// TIA Portal V20 export
FUNCTION_BLOCK "SysSensor"   // FB2040, FBD
TITLE = manage a sensor
{ S7_Optimized_Access := 'TRUE' }
AUTHOR : MiCROTEC
VERSION : 1.5
// -2021.12 : Martin / -2018.12 : Martin
// stored: AutoNumber false, MemoryReserve 100, SetENOAutomatically false
   VAR_INPUT
      errOccIn { ExternalAccessible := 'False'; ExternalVisible := 'False'; ExternalWritable := 'False'} : Bool;   // fault input (sensor signal or a combination of sensors)
      errOccVal { ExternalAccessible := 'False'; ExternalVisible := 'False'; ExternalWritable := 'False'} : Real;   // fault value for fault input
      errFreeIn { ExternalAccessible := 'False'; ExternalVisible := 'False'; ExternalWritable := 'False'} : Bool;   // fault input 2 (sensor signal or a combination of sensors)
      errFreeVal { ExternalAccessible := 'False'; ExternalVisible := 'False'; ExternalWritable := 'False'} : Real;   // fault value for fault input 2
      errCycleIn { ExternalAccessible := 'False'; ExternalVisible := 'False'; ExternalWritable := 'False'} : Bool;   // fault cycle input (this input increment a counter, counter is reset with rise or fallinge edge of sensor )
      errCycleVal { ExternalAccessible := 'False'; ExternalVisible := 'False'; ExternalWritable := 'False'} : Real;   // fault cycle value (if counter exceeds this value then error is set )
      sensor { ExternalAccessible := 'False'; ExternalVisible := 'False'; ExternalWritable := 'False'} : Bool;   // sensor signal
      enable { ExternalAccessible := 'False'; ExternalVisible := 'False'; ExternalWritable := 'False'} : Bool;   // if enable is true than the counter count, ex. run message from conv.
      ack { ExternalAccessible := 'False'; ExternalVisible := 'False'; ExternalWritable := 'False'} : Bool;   // acknowledg faults
      onDelVal { ExternalAccessible := 'False'; ExternalVisible := 'False'; ExternalWritable := 'False'} : Real;   // delayed on value for delayed on
      offDelVal { ExternalAccessible := 'False'; ExternalVisible := 'False'; ExternalWritable := 'False'} : Real;   // delayed off value for delayed off
      occOnVal { ExternalAccessible := 'False'; ExternalVisible := 'False'; ExternalWritable := 'False'} : Real;   // delayed on value for sensor occupied
      occOffVal { ExternalAccessible := 'False'; ExternalVisible := 'False'; ExternalWritable := 'False'} : Real;   // delayed off value for sensor occupied
      cntrVal { ExternalAccessible := 'False'; ExternalVisible := 'False'; ExternalWritable := 'False'} : Real;   // count value per cycle, if absolut encoder than activate "Param.AbsolutEncoder"
      absEnc { ExternalAccessible := 'False'; ExternalVisible := 'False'; ExternalWritable := 'False'} : Bool;   // activate absolut encoder for "countValue"
      reset { ExternalAccessible := 'False'; ExternalVisible := 'False'; ExternalWritable := 'False'} : Bool;   // reset the counter values and also the outputs
   END_VAR
   VAR_OUTPUT
      err { ExternalAccessible := 'False'; ExternalVisible := 'False'; ExternalWritable := 'False'} : Bool;   // Sensor fault , sensor is broken or is dirty
      errOcc { ExternalAccessible := 'False'; ExternalVisible := 'False'; ExternalWritable := 'False'} : Bool;   // Sensor fault , was to long occupied, maybe dirty or misaligned
      errFree { ExternalAccessible := 'False'; ExternalVisible := 'False'; ExternalWritable := 'False'} : Bool;   // Sensor fault , was to long free, maybe dirty or misaligned
      errCycle { ExternalAccessible := 'False'; ExternalVisible := 'False'; ExternalWritable := 'False'} : Bool;   // Sensor fault , plausibility check of cycles, after a certain amount(#errCycleVal) of trigger(#errCycleIn) the sensor had no rising or falling edge
      onDel { ExternalAccessible := 'False'; ExternalVisible := 'False'; ExternalWritable := 'False'} : Bool;   // sensor on delayed
      offDel { ExternalAccessible := 'False'; ExternalVisible := 'False'; ExternalWritable := 'False'} : Bool;   // sensor off delayed
      occ { ExternalAccessible := 'False'; ExternalVisible := 'False'; ExternalWritable := 'False'} : Bool;   // sensor occupied
      onCntr { ExternalAccessible := 'False'; ExternalVisible := 'False'; ExternalWritable := 'False'} : Real;   // counter for on delayed (if sensor is occupied it count, if free than reset)
      offCntr { ExternalAccessible := 'False'; ExternalVisible := 'False'; ExternalWritable := 'False'} : Real;   // counter for off delayed (if sensor is free it count, if occupied than reset)
      occOnCntr { ExternalAccessible := 'False'; ExternalVisible := 'False'; ExternalWritable := 'False'} : Real;   // on counter for occupied (if "occ" is "1" it count, if "0" than reset)
      occOffCntr { ExternalAccessible := 'False'; ExternalVisible := 'False'; ExternalWritable := 'False'} : Real;   // on counter for occupied (if "occ" is "0" it count, if "1" than reset)
   END_VAR
   VAR_IN_OUT
      Sen : "TypeSensor";
   END_VAR
   VAR
      var { ExternalAccessible := 'False'; ExternalVisible := 'False'; ExternalWritable := 'False'} : Struct
         "bool" : Bool;
         "byte" : Byte;
         "word" : Word;
         "dword" : DWord;
         "int" : Int;
         "dint" : DInt;
         "real" : Real;
         s5time : S5Time;
         "time" : Time;
         hm : Array[1..16] of Bool;
         fm : Array[1..16] of Bool;
      END_STRUCT;
      T { ExternalAccessible := 'False'; ExternalVisible := 'False'; ExternalWritable := 'False'} : Array[1..2] of IEC_TIMER;
      cntrValue { ExternalAccessible := 'False'; ExternalVisible := 'False'; ExternalWritable := 'False'} : Real;
      cntrValueOld { ExternalAccessible := 'False'; ExternalVisible := 'False'; ExternalWritable := 'False'} : Real;
      cntrErrOcc { ExternalAccessible := 'False'; ExternalVisible := 'False'; ExternalWritable := 'False'} : Real;   // counter for fault
      cntrErrFree { ExternalAccessible := 'False'; ExternalVisible := 'False'; ExternalWritable := 'False'} : Real;
      cntrErrCycle { ExternalAccessible := 'False'; ExternalVisible := 'False'; ExternalWritable := 'False'} : Real;
   END_VAR
   VAR_TEMP   // added for the SCL form of the ladder/FBD networks
      _w1 : Bool;
      _w2 : Bool;
      _w3 : Bool;
      _w4 : Bool;
   END_VAR
BEGIN

REGION Network 1: counter value value/perCycle or absolut encoder
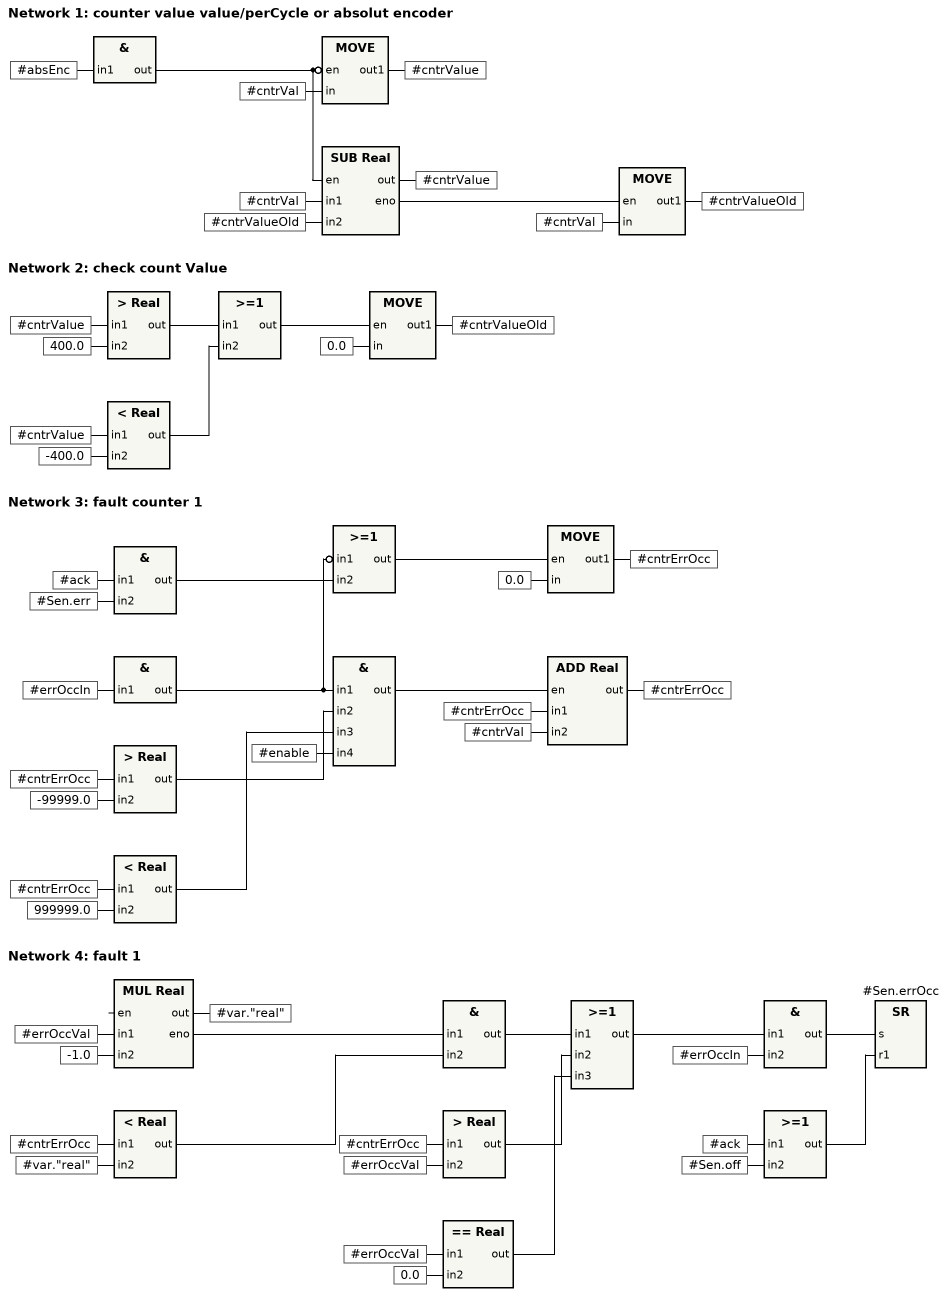
   // ENO of a box is taken as its EN; it also drops when the box reports an error
   IF NOT #absEnc THEN #cntrValue := #cntrVal; END_IF;
   IF #absEnc THEN
       #cntrValue := #cntrVal - #cntrValueOld;
       #cntrValueOld := #cntrVal;
   END_IF;
END_REGION

REGION Network 2: check count Value
   IF (#cntrValue > 400.0) OR (#cntrValue < (-400.0)) THEN #cntrValueOld := 0.0; END_IF;
END_REGION

REGION Network 3: fault counter 1
   IF NOT #errOccIn OR (#ack AND #Sen.err) THEN #cntrErrOcc := 0.0; END_IF;
   IF #errOccIn AND (#cntrErrOcc > (-99999.0)) AND (#cntrErrOcc < 999999.0) AND #enable THEN
       #cntrErrOcc := #cntrErrOcc + #cntrVal;
   END_IF;
END_REGION

REGION Network 4: fault 1
   // ENO of a box is taken as its EN; it also drops when the box reports an error
   #var."real" := #errOccVal * (-1.0);
   IF ((#cntrErrOcc < #var."real") OR (#cntrErrOcc > #errOccVal) OR (#errOccVal = 0.0)) AND #errOccIn THEN
       #Sen.errOcc := TRUE;   // SR flip-flop
   END_IF;
   IF #ack OR #Sen.off THEN #Sen.errOcc := FALSE; END_IF;
END_REGION

REGION Network 5: fault counter 2
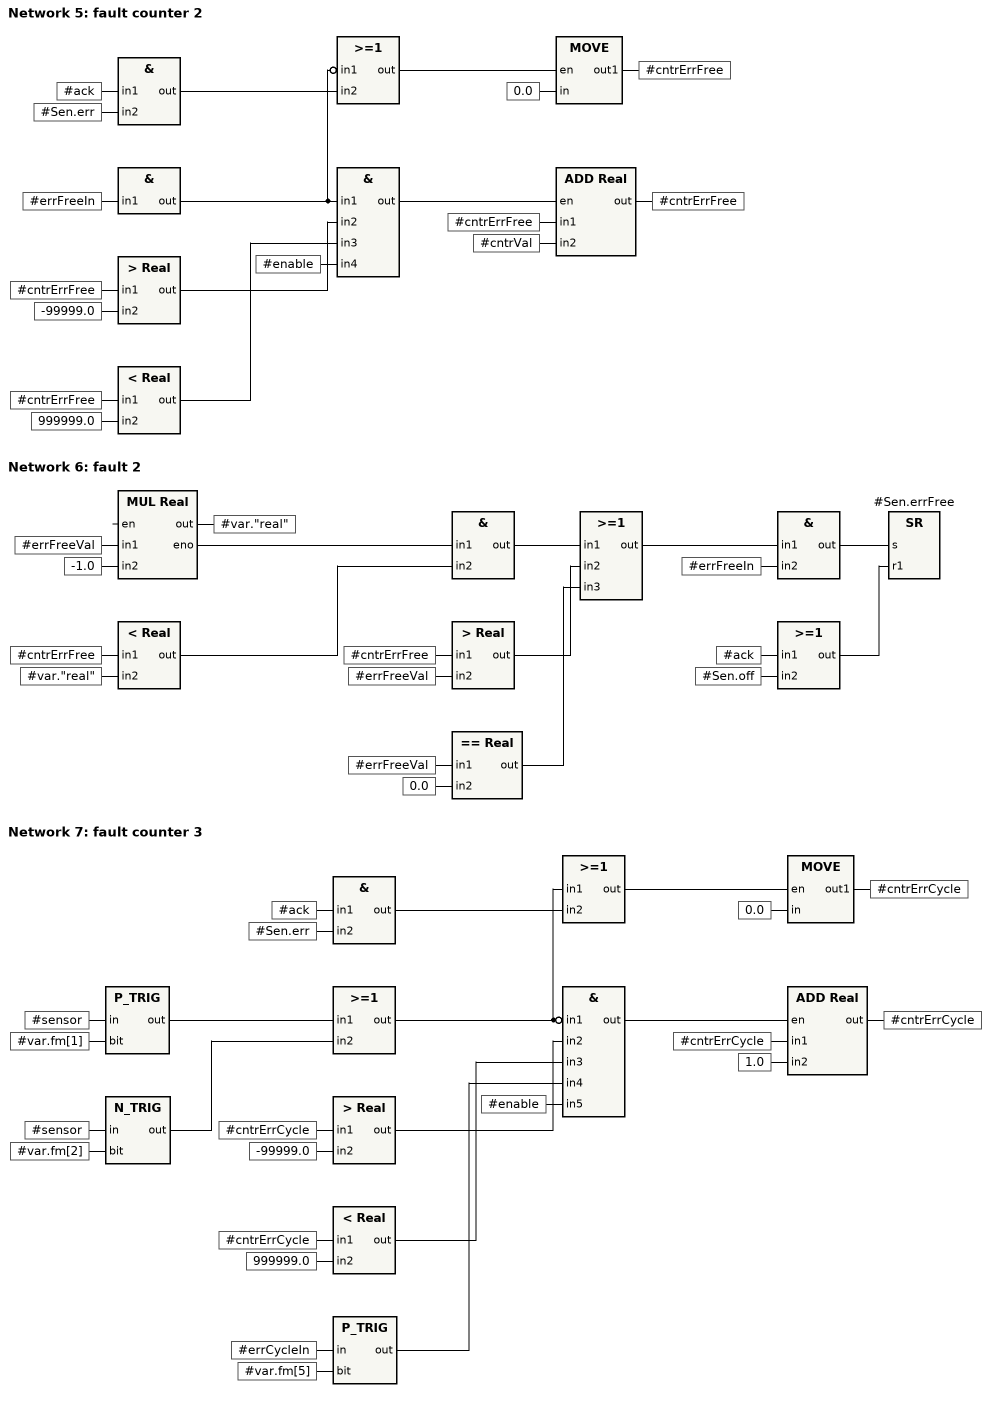
   IF NOT #errFreeIn OR (#ack AND #Sen.err) THEN #cntrErrFree := 0.0; END_IF;
   IF #errFreeIn AND (#cntrErrFree > (-99999.0)) AND (#cntrErrFree < 999999.0) AND #enable THEN
       #cntrErrFree := #cntrErrFree + #cntrVal;
   END_IF;
END_REGION

REGION Network 6: fault 2
   // ENO of a box is taken as its EN; it also drops when the box reports an error
   #var."real" := #errFreeVal * (-1.0);
   IF ((#cntrErrFree < #var."real") OR (#cntrErrFree > #errFreeVal) OR (#errFreeVal = 0.0)) AND #errFreeIn THEN
       #Sen.errFree := TRUE;   // SR flip-flop
   END_IF;
   IF #ack OR #Sen.off THEN #Sen.errFree := FALSE; END_IF;
END_REGION

REGION Network 7: fault counter 3
   #_w1 := #sensor AND NOT #var.fm[1];   // rising edge
   #var.fm[1] := #sensor;
   #_w2 := NOT #sensor AND #var.fm[2];   // falling edge
   #var.fm[2] := #sensor;
   #_w3 := #_w1 OR #_w2;
   IF #_w3 OR (#ack AND #Sen.err) THEN #cntrErrCycle := 0.0; END_IF;
   #_w4 := #errCycleIn AND NOT #var.fm[5];   // rising edge
   #var.fm[5] := #errCycleIn;
   IF NOT #_w3 AND (#cntrErrCycle > (-99999.0)) AND (#cntrErrCycle < 999999.0) AND #_w4 AND #enable THEN
       #cntrErrCycle := #cntrErrCycle + 1.0;
   END_IF;
END_REGION

REGION Network 8: fault 3
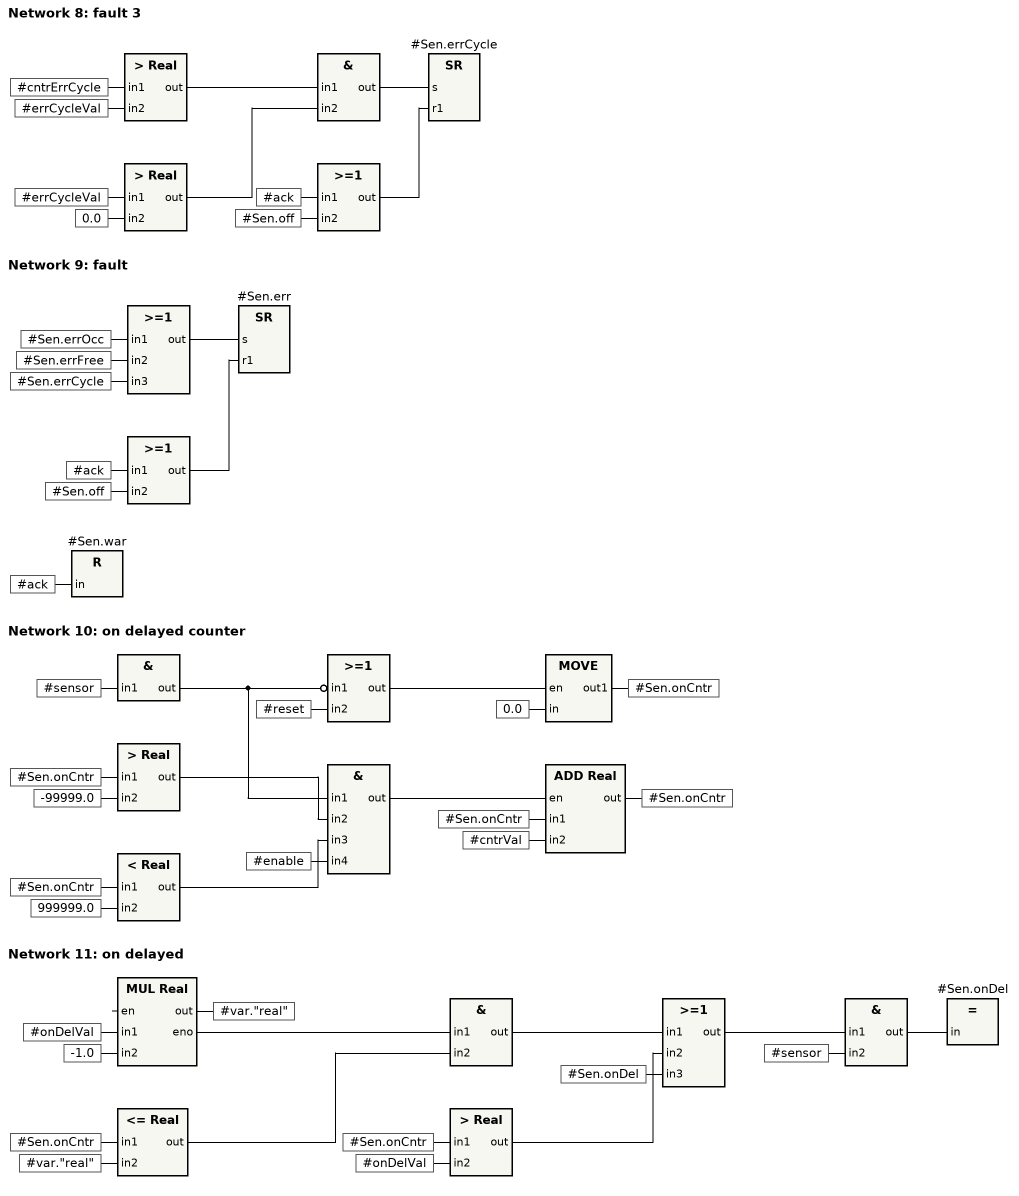
   IF (#cntrErrCycle > #errCycleVal) AND (#errCycleVal > 0.0) THEN
       #Sen.errCycle := TRUE;   // SR flip-flop
   END_IF;
   IF #ack OR #Sen.off THEN #Sen.errCycle := FALSE; END_IF;
END_REGION

REGION Network 9: fault
   IF #Sen.errOcc OR #Sen.errFree OR #Sen.errCycle THEN
       #Sen.err := TRUE;   // SR flip-flop
   END_IF;
   IF #ack OR #Sen.off THEN #Sen.err := FALSE; END_IF;
   IF #ack THEN #Sen.war := FALSE; END_IF;
END_REGION

REGION Network 10: on delayed counter
   IF NOT #sensor OR #reset THEN #Sen.onCntr := 0.0; END_IF;
   IF #sensor AND (#Sen.onCntr > (-99999.0)) AND (#Sen.onCntr < 999999.0) AND #enable THEN
       #Sen.onCntr := #Sen.onCntr + #cntrVal;
   END_IF;
END_REGION

REGION Network 11: on delayed
   // ENO of a box is taken as its EN; it also drops when the box reports an error
   #var."real" := #onDelVal * (-1.0);
   #Sen.onDel := ((#Sen.onCntr <= #var."real") OR (#Sen.onCntr > #onDelVal) OR #Sen.onDel) AND #sensor;
END_REGION

REGION Network 12: off delayed counter
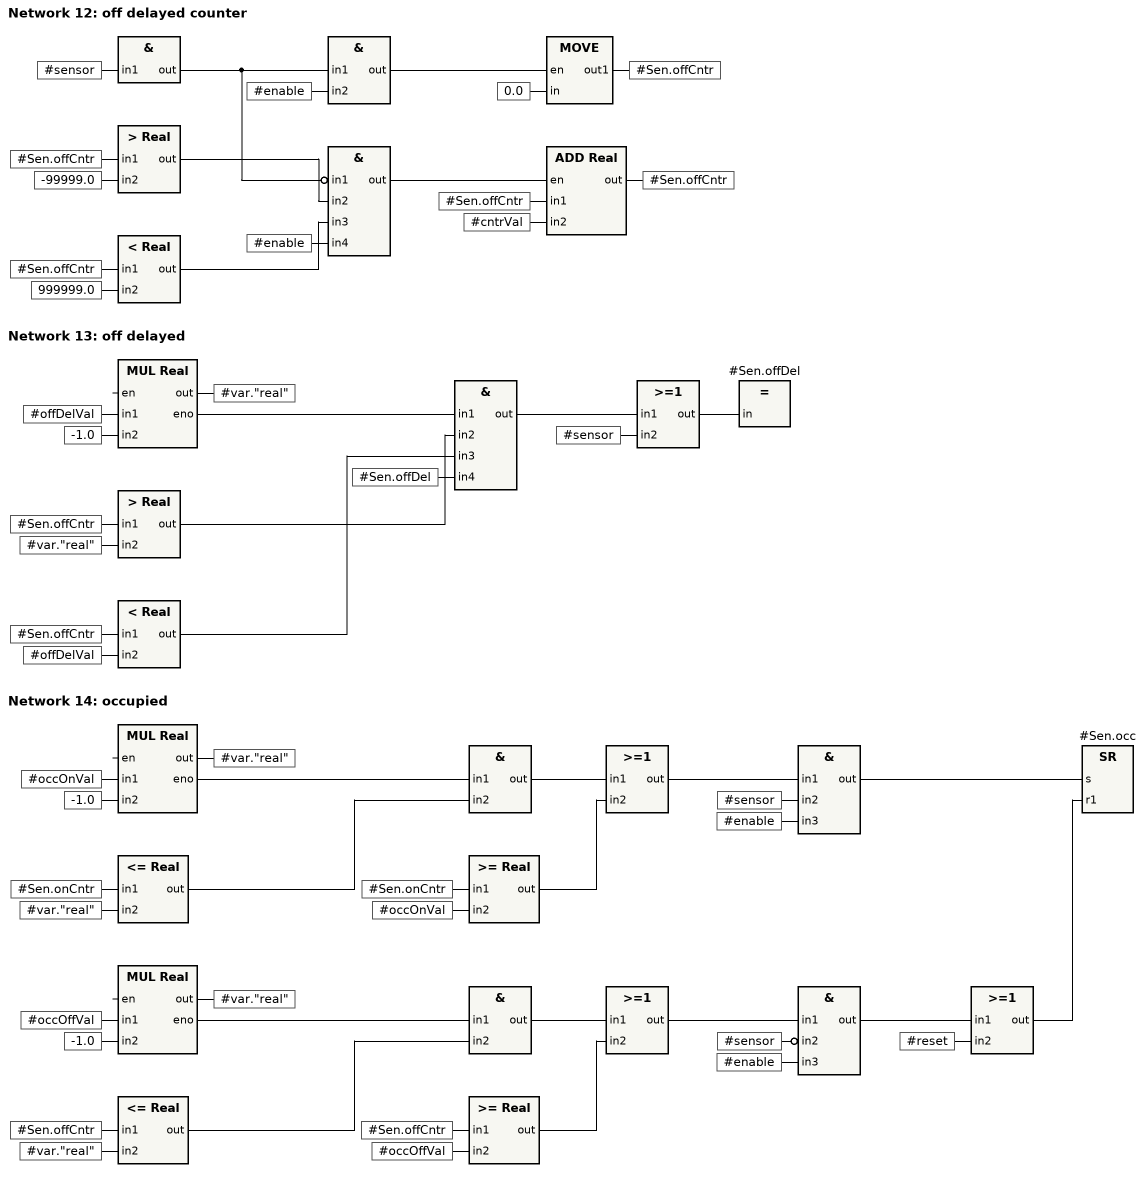
   IF #sensor AND #enable THEN #Sen.offCntr := 0.0; END_IF;
   IF NOT #sensor AND (#Sen.offCntr > (-99999.0)) AND (#Sen.offCntr < 999999.0) AND #enable THEN
       #Sen.offCntr := #Sen.offCntr + #cntrVal;
   END_IF;
END_REGION

REGION Network 13: off delayed
   // ENO of a box is taken as its EN; it also drops when the box reports an error
   #var."real" := #offDelVal * (-1.0);
   #Sen.offDel := ((#Sen.offCntr > #var."real") AND (#Sen.offCntr < #offDelVal) AND #Sen.offDel) OR #sensor;
END_REGION

REGION Network 14: occupied
   // ENO of a box is taken as its EN; it also drops when the box reports an error
   #var."real" := #occOnVal * (-1.0);
   #_w1 := ((#Sen.onCntr <= #var."real") OR (#Sen.onCntr >= #occOnVal)) AND #sensor AND #enable;
   #var."real" := #occOffVal * (-1.0);
   IF #_w1 THEN
       #Sen.occ := TRUE;   // SR flip-flop
   END_IF;
   IF (((#Sen.offCntr <= #var."real") OR (#Sen.offCntr >= #occOffVal)) AND NOT #sensor AND #enable) OR #reset THEN
       #Sen.occ := FALSE;
   END_IF;
END_REGION

REGION Network 15: positive / negative edge
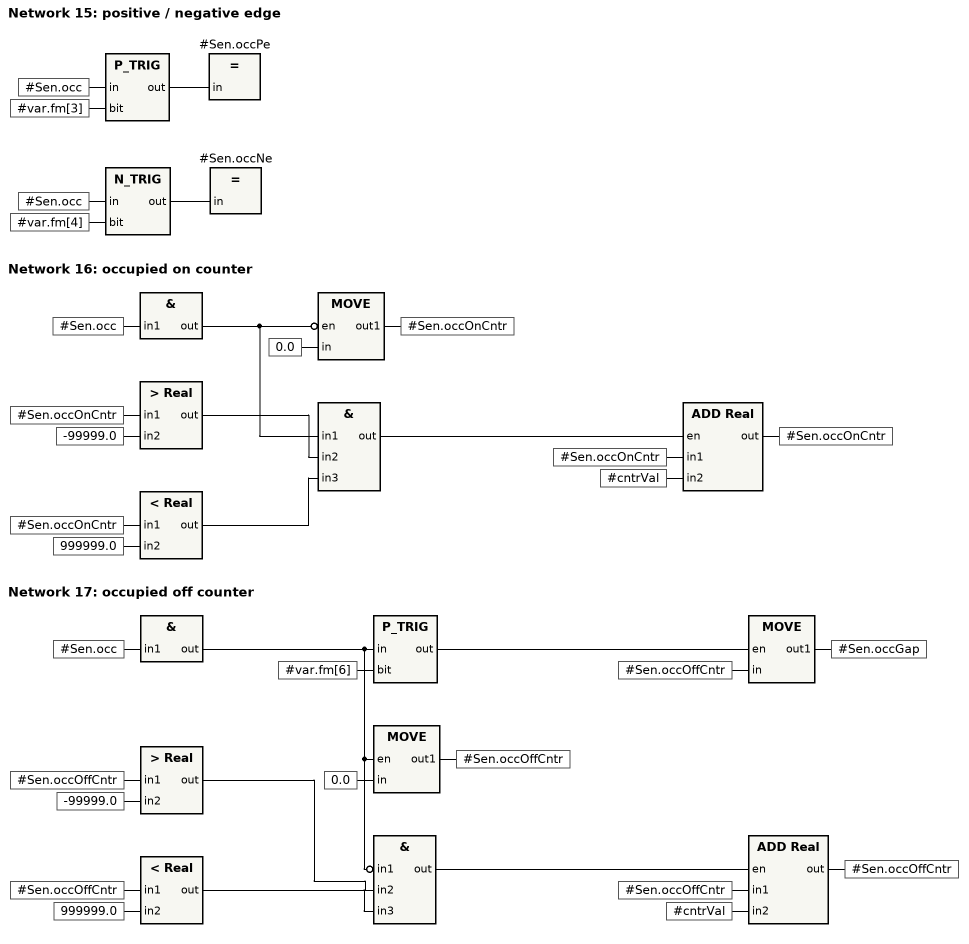
   #_w1 := #Sen.occ AND NOT #var.fm[3];   // rising edge
   #var.fm[3] := #Sen.occ;
   #Sen.occPe := #_w1;
   #_w2 := NOT #Sen.occ AND #var.fm[4];   // falling edge
   #var.fm[4] := #Sen.occ;
   #Sen.occNe := #_w2;
END_REGION

REGION Network 16: occupied on counter
   IF NOT #Sen.occ THEN #Sen.occOnCntr := 0.0; END_IF;
   IF #Sen.occ AND (#Sen.occOnCntr > (-99999.0)) AND (#Sen.occOnCntr < 999999.0) THEN
       #Sen.occOnCntr := #Sen.occOnCntr + #cntrVal;
   END_IF;
END_REGION

REGION Network 17: occupied off counter
   #_w1 := #Sen.occ AND NOT #var.fm[6];   // rising edge
   #var.fm[6] := #Sen.occ;
   IF #_w1 THEN #Sen.occGap := #Sen.occOffCntr; END_IF;
   IF #Sen.occ THEN #Sen.occOffCntr := 0.0; END_IF;
   IF NOT #Sen.occ AND (#Sen.occOffCntr > (-99999.0)) AND (#Sen.occOffCntr < 999999.0) THEN
       #Sen.occOffCntr := #Sen.occOffCntr + #cntrVal;
   END_IF;
END_REGION

REGION Network 18 (SCL): write outputs
      #err := #Sen.err;
       #errOcc := #Sen.errOcc;
       #errFree := #Sen.errFree;
       #errCycle := #Sen.errCycle;
       #onDel :=  #Sen.onDel;
       #offDel :=  #Sen.offDel;
       #occ := #Sen.occ;
       #onCntr :=  #Sen.onCntr;
       #offCntr := #Sen.offCntr;
       #occOnCntr :=    #Sen.occOnCntr ;
       #occOffCntr :=  #Sen.occOffCntr;

       #Sen.sen := #sensor;
END_REGION
END_FUNCTION_BLOCK
